(* Schneider Machine Expert - Basic project CApture Network Traffic With Timer, file version 1.6.0.0 *)
(* ProjectInformations: Name=New project *)

HARDWARE
  Cpu 0: TM221CE16R
  EthernetConfiguration: NetworkName=M221, IpAllocationMode=FixedAddress, IpAddress=0.0.0.0, SubnetMask=0.0.0.0
  SerialLineConfiguration: Baud=Baud19200, Parity=ParityEven, DataBits=DataBits8, StopBits=StopBits1, PhysicalMedium=PhysicalMediumRs485, TransmissionMode=TransmissionModeModbusRtu, SlaveId=1, Addressing=SlaveAddressing
  MastTask: UsePeriodScanMode=false, PeriodScan=100
  FastTask: Period=255
  CpuBehavior: StartingMode=StartAsPreviousState, AutoSaveRamOnEeprom=true, WatchdogPeriod=250

SYMBOLS  (address, symbol, comment, settings)
  %TM0        [Preset=1211, Base=OneSecond]
  %TM1        [Preset=2347, Base=OneSecond]

POU New POU
  (* SectionNumber=1 *)

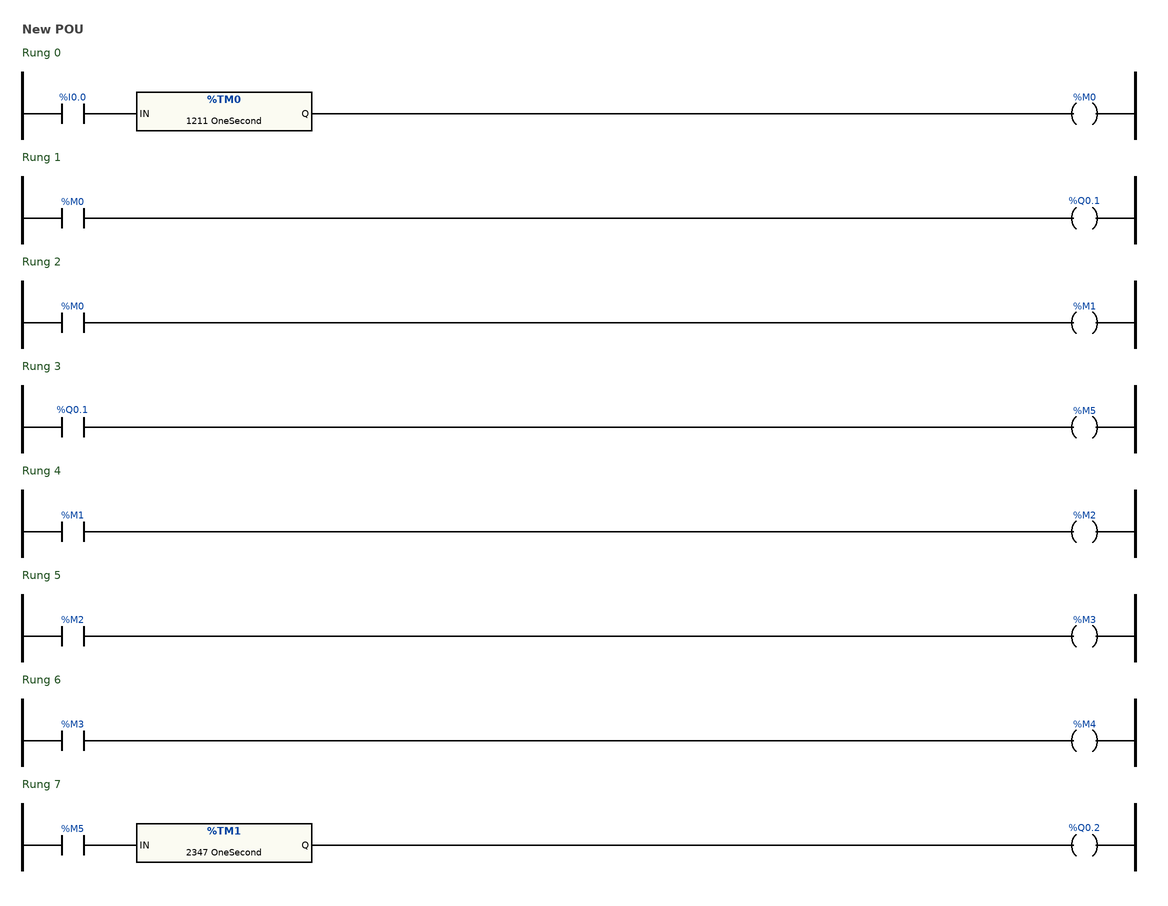

// Rung 0
  BLK %TM0
  LD %I0.0
  IN
  OUT_BLK
  LD Q
  ST %M0
  END_BLK
  // as ST:
  //   %TM0(IN := %I0.0);
  //   %M0 := %TM0.Q;

// Rung 1
  LD %M0
  ST %Q0.1
  // as ST:
  //   %Q0.1 := %M0;

// Rung 2
  LD %M0
  ST %M1
  // as ST:
  //   %M1 := %M0;

// Rung 3
  LD %Q0.1
  ST %M5
  // as ST:
  //   %M5 := %Q0.1;

// Rung 4
  LD %M1
  ST %M2
  // as ST:
  //   %M2 := %M1;

// Rung 5
  LD %M2
  ST %M3
  // as ST:
  //   %M3 := %M2;

// Rung 6
  LD %M3
  ST %M4
  // as ST:
  //   %M4 := %M3;

// Rung 7
  BLK %TM1
  LD %M5
  IN
  OUT_BLK
  LD Q
  ST %Q0.2
  END_BLK
  // as ST:
  //   %TM1(IN := %M5);
  //   %Q0.2 := %TM1.Q;
